FUNCTION_BLOCK CMP_OC_DINT
VAR_INPUT
	BOOL_INTERLOCK : BOOL; (*INTERLOCK*)
	DINT_1: DINT;		(*WORD 1*)
	END_VAR


VAR_OUTPUT
	BZ_OUTPUT_BOOL : BOOL;
END_VAR


VAR
	OUT_1: BOOL;
END_VAR

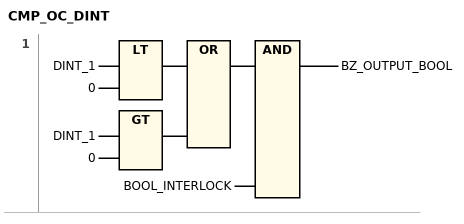
// NETWORK 1
BZ_OUTPUT_BOOL := (DINT_1 < 0 OR DINT_1 > 0) AND BOOL_INTERLOCK;

END_FUNCTION_BLOCK

(* stored: Version 1.1.0.1, ProductVersion 3.1.4024.12
   POU CMP_OC_DINT: Id {a785ee68-f1b8-479d-bb80-501a6005d404}, SpecialFunc None *)
